// SIMATIC S7-200 project (STEP 7-Micro/WIN), CPU 226 CN REL 02.01

ORGANIZATION_BLOCK MAIN:OB1
TITLE=PROGRAM COMMENTS
BEGIN
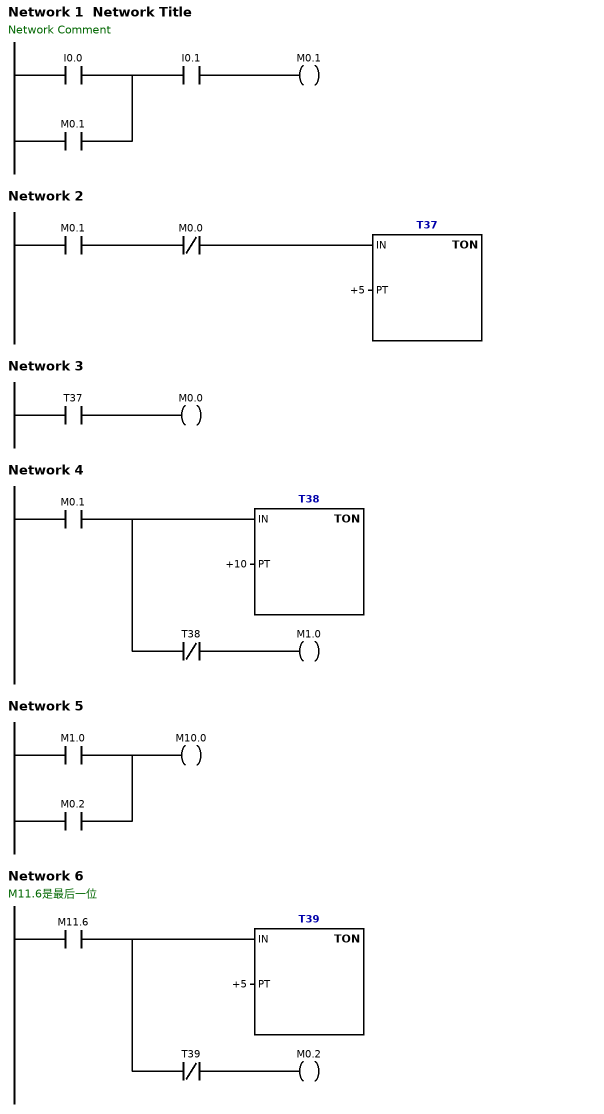
Network 1 // Network Title
// Network Comment
LD     I0.0
O      M0.1
A      I0.1
=      M0.1
Network 2
LD     M0.1
AN     M0.0
TON    T37, +5
Network 3
LD     T37
=      M0.0
Network 4
LD     M0.1
TON    T38, +10
AN     T38
=      M1.0
Network 5
LD     M1.0
O      M0.2
=      M10.0
Network 6
// M11.6是最后一位
LD     M11.6
TON    T39, +5
AN     T39
=      M0.2
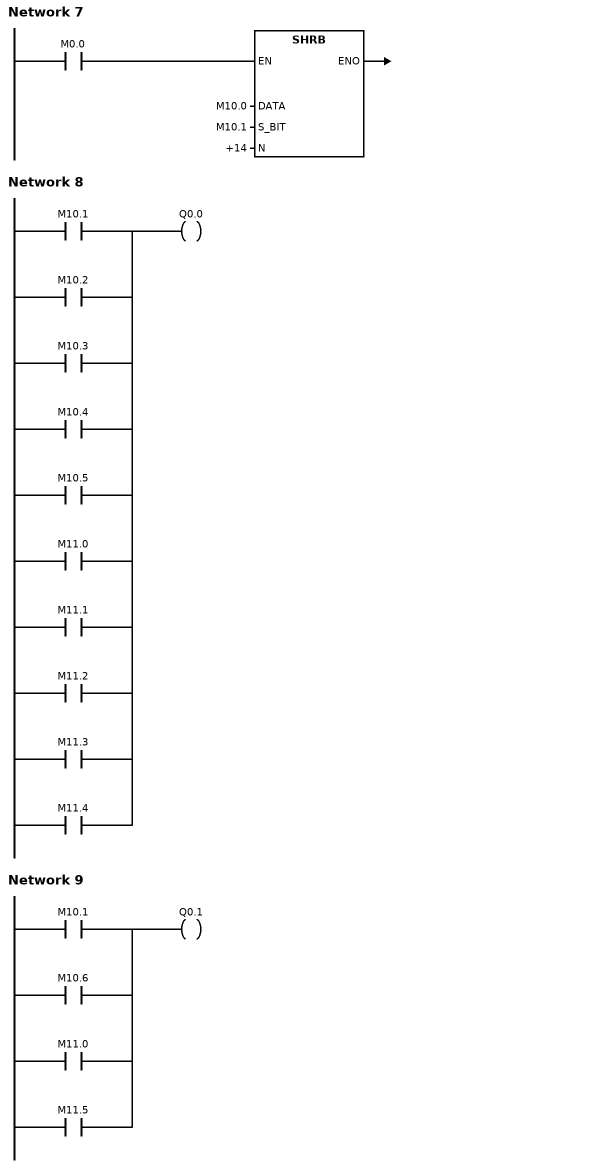
Network 7
LD     M0.0
SHRB   M10.0, M10.1, +14
Network 8
LD     M10.1
O      M10.2
O      M10.3
O      M10.4
O      M10.5
O      M11.0
O      M11.1
O      M11.2
O      M11.3
O      M11.4
=      Q0.0
Network 9
LD     M10.1
O      M10.6
O      M11.0
O      M11.5
=      Q0.1
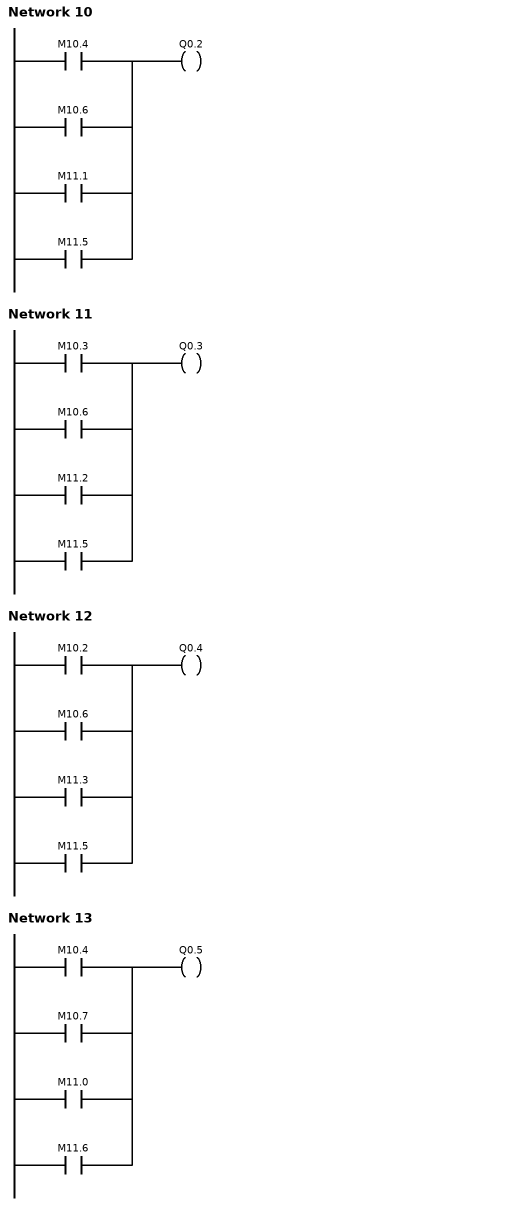
Network 10
LD     M10.4
O      M10.6
O      M11.1
O      M11.5
=      Q0.2
Network 11
LD     M10.3
O      M10.6
O      M11.2
O      M11.5
=      Q0.3
Network 12
LD     M10.2
O      M10.6
O      M11.3
O      M11.5
=      Q0.4
Network 13
LD     M10.4
O      M10.7
O      M11.0
O      M11.6
=      Q0.5
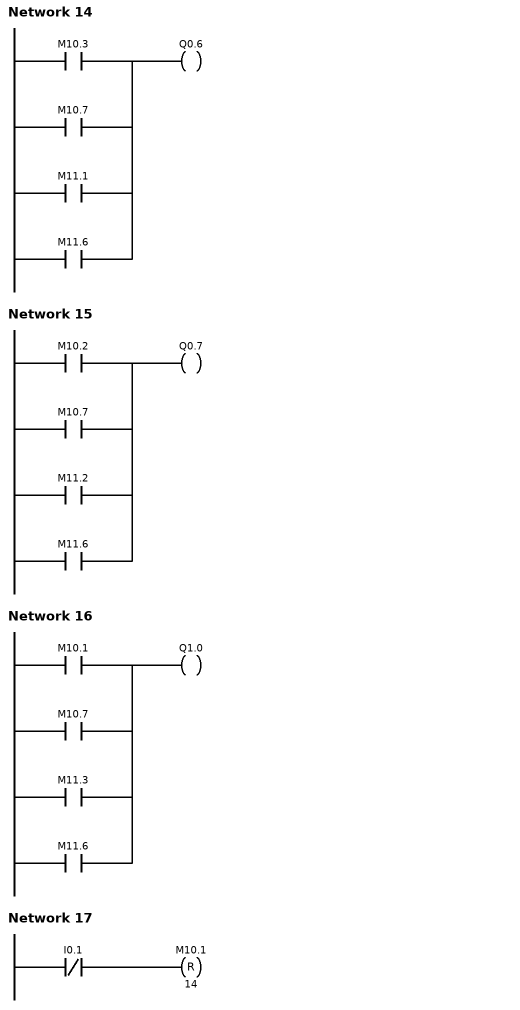
Network 14
LD     M10.3
O      M10.7
O      M11.1
O      M11.6
=      Q0.6
Network 15
LD     M10.2
O      M10.7
O      M11.2
O      M11.6
=      Q0.7
Network 16
LD     M10.1
O      M10.7
O      M11.3
O      M11.6
=      Q1.0
Network 17
LDN    I0.1
R      M10.1, 14
END_ORGANIZATION_BLOCK
